TYPE ST_EX260Io :
STRUCT
	State 	AT %I* : UINT;
	Ctrl 	AT %Q* : UINT;
	In0 	AT %I* : SINT;
	In1 	AT %I* : SINT;
	Out0 	AT %Q* : BYTE;
	Out1 	AT %Q* : BYTE;
	Out2 	AT %Q* : BYTE;
	Out3 	AT %Q* : BYTE;
END_STRUCT
END_TYPE

(* stored: Version 1.1.0.1
   DUT ST_EX260Io: Id {2bd75630-0ef5-465d-a5c0-af6587498ff2} *)
